// TIA Portal project "Treino_com_Variaveis_Arrays_structs" (V14)

(* hardware
DEVICE "S7-1200 station_1"  S7-1200 Station
   slot 0: "Rack_0"  S7-1200 Rack  Rack  V1.0
   slot 1: "PLC_1"  CPU 1214C DC/DC/DC  6ES7 214-1AG40-0XB0  V4.2
*)

// ===== PLC "PLC_1"  CPU 1214C DC/DC/DC =====

DATA_BLOCK "Motor"   // DB1
{ S7_Optimized_Access := 'TRUE' }
VERSION : 0.1
   VAR
      MotorClass : Struct
         Ligado : Bool := 1;
         Nome : String[10] := 'Bomba01';
         Velocidade : Int := 1735;
         Temperatura : Real := 22.5;
         TempoFuncionamento : Time := T#1000ms;
         NumeroCiclos : DInt := 1000000;
         StatusMotor : Byte := 16#03;
      END_STRUCT;
      Motores : Array[1..5] of Struct
      END_STRUCT;
   END_VAR
BEGIN
END_DATA_BLOCK

ORGANIZATION_BLOCK "Main"   // OB1, LAD, ProgramCycle
TITLE = "Main Program Sweep (Cycle)"
{ S7_Optimized_Access := 'TRUE' }
VERSION : 0.1
   VAR_INPUT
      Initial_Call : Bool;   // Initial call of this OB
      Remanence : Bool;   // =True, if remanent data are available
   END_VAR
BEGIN
END_ORGANIZATION_BLOCK